// Variables to be accessed by Labview or PC.
VAR_GLOBAL
END_VAR

(* stored: Version 1.1.0.1, ProductVersion 3.1.4022.18
   GVL PC: Id {384e0a86-f692-4694-a993-0166314ad626} *)
